FUNCTION_BLOCK DisableConveyor (* Basic Function Block Type *)
  (* Standard: 61499-2 *)
  (* Version 0.0, 4/12/2016, Aalto_IT, nxtControl GmbH, Template *)
  PACKAGE Main;
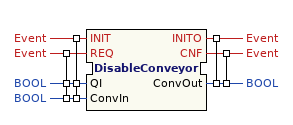
  EVENT_INPUT
    INIT WITH QI, ConvIn; (* Initialization Request *)
    REQ WITH QI, ConvIn; (* Normal Execution Request *)
  END_EVENT
  EVENT_OUTPUT
    INITO WITH ConvOut; (* Initialization Confirm *)
    CNF WITH ConvOut; (* Execution Confirmation *)
  END_EVENT
  VAR_INPUT
    QI : BOOL;
    ConvIn : BOOL; (* Input event qualifier *)
  END_VAR
  VAR_OUTPUT
    ConvOut : BOOL; (* Output event qualifier *)
  END_VAR
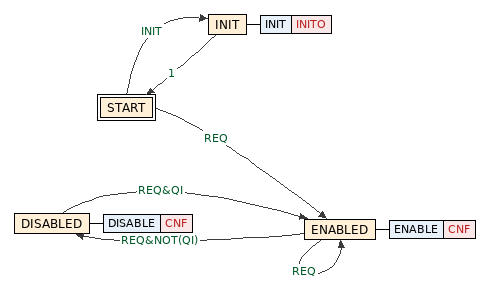
  EC_STATES
    START; (* Initial State *)
    INIT : INIT -> INITO; (* Initialization *)
    ENABLED : ENABLE -> CNF; (* Normal execution *)
    DISABLED : DISABLE -> CNF; (* Normal execution *)
  END_STATES
  EC_TRANSITIONS
    START TO INIT := INIT;
    INIT TO START := 1;
    ENABLED TO DISABLED := REQ&NOT(QI);
    START TO ENABLED := REQ;
    DISABLED TO ENABLED := REQ&QI;
    ENABLED TO ENABLED := REQ;
  END_TRANSITIONS
  ALGORITHM INIT IN ST: (* Initialization algorithm *)
;
  END_ALGORITHM
  ALGORITHM ENABLE IN ST: (* Normally executed algorithm *)
;
ConvOut:=ConvIn;
  END_ALGORITHM
  ALGORITHM DISABLE IN ST:
;
ConvOut:=FALSE;
  END_ALGORITHM
END_FUNCTION_BLOCK
